{attribute 'GeneratedUsingTerminal: EL3204-0200-0016'}
{attribute addProperty BoxType "EL3204-0200-0016"}
{attribute addProperty Id "EtcSlaveTerminalBaseRTD_Inputs_Channel_1AT %I*RTD_Inputs_Channel_9575FEA17RTD_Inputs_Channel_2AT %I*RTD_Inputs_Channel_9575FEA17RTD_Inputs_Channel_3AT %I*RTD_Inputs_Channel_9575FEA17RTD_Inputs_Channel_4AT %I*RTD_Inputs_Channel_9575FEA17WcStateAT %I*WcState_9091E0EB2InfoDataAT %I*InfoData_32EB74EA10"}
{attribute addProperty CRC "2951308367"}
{attribute addProperty Size "40"}
TYPE EL3204_AFE9644F EXTENDS EtcSlaveTerminalBase :
STRUCT
	{attribute addProperty Name "RTD_Inputs_Channel_1"}
	RTD_Inputs_Channel_1 : RTD_Inputs_Channel_9575FEA1;
	{attribute addProperty Name "RTD_Inputs_Channel_2"}
	RTD_Inputs_Channel_2 : RTD_Inputs_Channel_9575FEA1;
	{attribute addProperty Name "RTD_Inputs_Channel_3"}
	RTD_Inputs_Channel_3 : RTD_Inputs_Channel_9575FEA1;
	{attribute addProperty Name "RTD_Inputs_Channel_4"}
	RTD_Inputs_Channel_4 : RTD_Inputs_Channel_9575FEA1;
	{attribute addProperty Name "WcState"}
	WcState : WcState_9091E0EB;
	{attribute addProperty Name "InfoData"}
	InfoData : InfoData_32EB74EA;
END_STRUCT
END_TYPE

(* stored: Version 1.2.0.0, ProductVersion 3.1.4024.9
   DUT EL3204_AFE9644F: Id {2177c9e0-7157-43a8-9804-ac670da37fbd} *)
